// TwinCAT 3 PLC project PlcProj
// ProgramVersion: 3.1.4023.0
// libraries:
//   Tc2_Standard, * (Beckhoff Automation GmbH)
//   Tc2_System, * (Beckhoff Automation GmbH)
//   Tc3_Module, * (Beckhoff Automation GmbH)
// project tree:
//   DUTs/ stChild.TcDUT, stMain.TcDUT
//   GVLs/ GVL.TcGVL
//   / PlcTask.TcTTO
//   POUs/ MAIN.TcPOU
// real-time tasks:
//   TASK PlcTask: cycle T#10ms, priority 20, ADS port 350

CONFIGURATION PlcProj
    RESOURCE PLC ON TwinCAT3
        TASK PlcTask(INTERVAL := T#10ms, PRIORITY := 20);
        PROGRAM MAIN WITH PlcTask : MAIN;
    END_RESOURCE
END_CONFIGURATION

// ---- DUTs/stChild.TcDUT
TYPE stChild :
	STRUCT
		fVar1 : LREAL;
		fVar2 : REAL;
		nVar3 : WORD;
	END_STRUCT
END_TYPE

// ---- DUTs/stMain.TcDUT
TYPE stMain :
	STRUCT
		bVar1 : BOOL;
		bVar2 : BOOL;
		fVar3 : LREAL;
		fVar4 : REAL;
		nVar5 : INT;
		nVar6 : DINT;
		nVar7 : stChild;
	END_STRUCT
END_TYPE

// ---- GVLs/GVL.TcGVL
{attribute 'qualified_only'}
VAR_GLOBAL
	ST_Dat1 : stMain;
	ST_Dat2 : stMain;
END_VAR

// ---- POUs/MAIN.TcPOU
PROGRAM MAIN
VAR
	randomValue : LREAL;
	Rand: DRAND;
END_VAR

Rand(Seed:=0,Num=>randomValue);

GVL.ST_Dat1.bVar1:=INT_TO_BOOL(LREAL_TO_INT(randomValue));
GVL.ST_Dat1.bVar2:=NOT INT_TO_BOOL(LREAL_TO_INT(randomValue));
GVL.ST_Dat1.fVar3:=randomValue*1;
GVL.ST_Dat1.fVar4:=LREAL_TO_REAL(randomValue*2);
GVL.ST_Dat1.nVar5:=LREAL_TO_INT(randomValue*3);
GVL.ST_Dat1.nVar6:=LREAL_TO_INT(randomValue*4);
GVL.ST_Dat1.nVar7.fVar1:=randomValue*5;
GVL.ST_Dat1.nVar7.fVar2:=LREAL_TO_REAL(randomValue*6);
GVL.ST_Dat1.nVar7.nVar3:=LREAL_TO_WORD(randomValue*100);

GVL.ST_Dat2.bVar1:=INT_TO_BOOL(LREAL_TO_INT(randomValue));
GVL.ST_Dat2.bVar2:=NOT INT_TO_BOOL(LREAL_TO_INT(randomValue));
GVL.ST_Dat2.fVar3:=randomValue*1;;
GVL.ST_Dat2.fVar4:=LREAL_TO_REAL(randomValue*2);
GVL.ST_Dat2.nVar5:=LREAL_TO_INT(randomValue*3);
GVL.ST_Dat2.nVar6:=LREAL_TO_INT(randomValue*4);
GVL.ST_Dat2.nVar7.fVar1:=randomValue*5;
GVL.ST_Dat2.nVar7.fVar2:=LREAL_TO_REAL(randomValue*6);
GVL.ST_Dat2.nVar7.nVar3:=LREAL_TO_WORD(randomValue*100);

END_PROGRAM
